// TIA Portal V19 export
FUNCTION "OUTPUT" : Void   // FC2, LAD
{ S7_Optimized_Access := 'TRUE' }
// stored: SetENOAutomatically false
BEGIN

REGION Network 1: "MFG FEED PUMP OP"
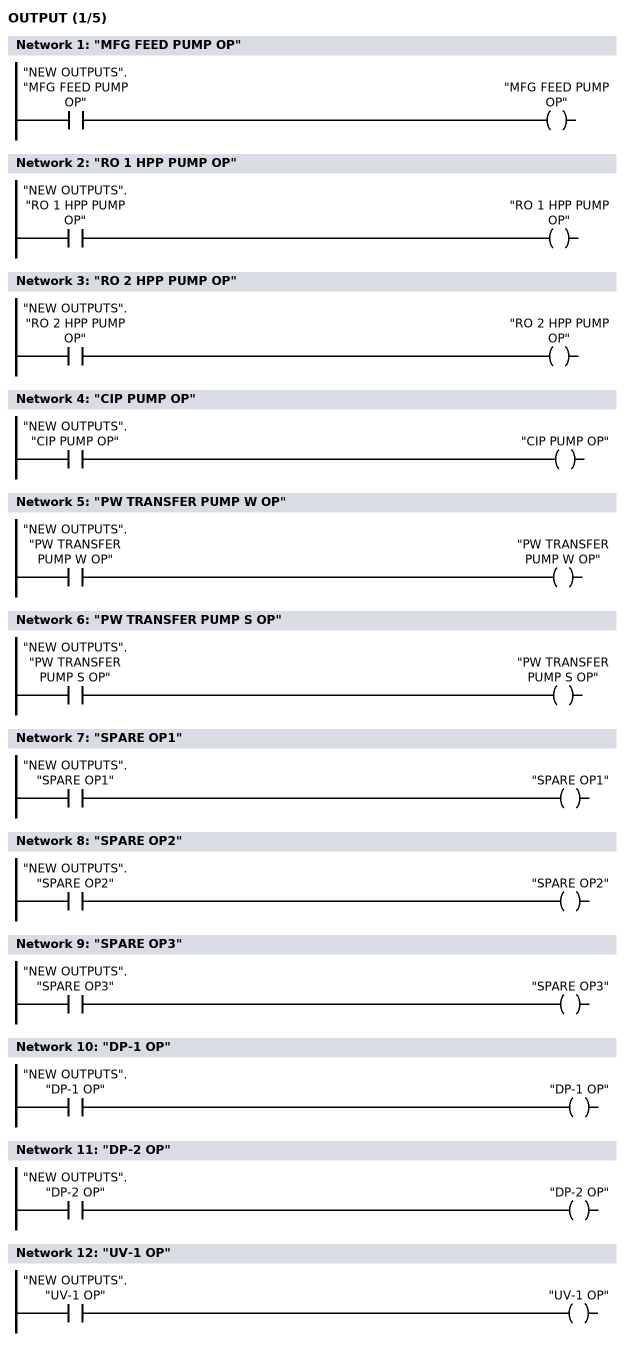
   RUNG wire#powerrail
      Contact( "NEW OUTPUTS"."MFG FEED PUMP OP" )
      Coil( "MFG FEED PUMP OP" )
   END_RUNG
   // the same network as SCL:
   "MFG FEED PUMP OP" := "NEW OUTPUTS"."MFG FEED PUMP OP";
END_REGION

REGION Network 2: "RO 1 HPP PUMP OP"
   RUNG wire#powerrail
      Contact( "NEW OUTPUTS"."RO 1 HPP PUMP OP" )
      Coil( "RO 1 HPP PUMP OP" )
   END_RUNG
   // the same network as SCL:
   "RO 1 HPP PUMP OP" := "NEW OUTPUTS"."RO 1 HPP PUMP OP";
END_REGION

REGION Network 3: "RO 2 HPP PUMP OP"
   RUNG wire#powerrail
      Contact( "NEW OUTPUTS"."RO 2 HPP PUMP OP" )
      Coil( "RO 2 HPP PUMP OP" )
   END_RUNG
   // the same network as SCL:
   "RO 2 HPP PUMP OP" := "NEW OUTPUTS"."RO 2 HPP PUMP OP";
END_REGION

REGION Network 4: "CIP PUMP OP"
   RUNG wire#powerrail
      Contact( "NEW OUTPUTS"."CIP PUMP OP" )
      Coil( "CIP PUMP OP" )
   END_RUNG
   // the same network as SCL:
   "CIP PUMP OP" := "NEW OUTPUTS"."CIP PUMP OP";
END_REGION

REGION Network 5: "PW TRANSFER PUMP W OP"
   RUNG wire#powerrail
      Contact( "NEW OUTPUTS"."PW TRANSFER PUMP W OP" )
      Coil( "PW TRANSFER PUMP W OP" )
   END_RUNG
   // the same network as SCL:
   "PW TRANSFER PUMP W OP" := "NEW OUTPUTS"."PW TRANSFER PUMP W OP";
END_REGION

REGION Network 6: "PW TRANSFER PUMP S OP"
   RUNG wire#powerrail
      Contact( "NEW OUTPUTS"."PW TRANSFER PUMP S OP" )
      Coil( "PW TRANSFER PUMP S OP" )
   END_RUNG
   // the same network as SCL:
   "PW TRANSFER PUMP S OP" := "NEW OUTPUTS"."PW TRANSFER PUMP S OP";
END_REGION

REGION Network 7: "SPARE OP1"
   RUNG wire#powerrail
      Contact( "NEW OUTPUTS"."SPARE OP1" )
      Coil( "SPARE OP1" )
   END_RUNG
   // the same network as SCL:
   "SPARE OP1" := "NEW OUTPUTS"."SPARE OP1";
END_REGION

REGION Network 8: "SPARE OP2"
   RUNG wire#powerrail
      Contact( "NEW OUTPUTS"."SPARE OP2" )
      Coil( "SPARE OP2" )
   END_RUNG
   // the same network as SCL:
   "SPARE OP2" := "NEW OUTPUTS"."SPARE OP2";
END_REGION

REGION Network 9: "SPARE OP3"
   RUNG wire#powerrail
      Contact( "NEW OUTPUTS"."SPARE OP3" )
      Coil( "SPARE OP3" )
   END_RUNG
   // the same network as SCL:
   "SPARE OP3" := "NEW OUTPUTS"."SPARE OP3";
END_REGION

REGION Network 10: "DP-1 OP"
   RUNG wire#powerrail
      Contact( "NEW OUTPUTS"."DP-1 OP" )
      Coil( "DP-1 OP" )
   END_RUNG
   // the same network as SCL:
   "DP-1 OP" := "NEW OUTPUTS"."DP-1 OP";
END_REGION

REGION Network 11: "DP-2 OP"
   RUNG wire#powerrail
      Contact( "NEW OUTPUTS"."DP-2 OP" )
      Coil( "DP-2 OP" )
   END_RUNG
   // the same network as SCL:
   "DP-2 OP" := "NEW OUTPUTS"."DP-2 OP";
END_REGION

REGION Network 12: "UV-1 OP"
   RUNG wire#powerrail
      Contact( "NEW OUTPUTS"."UV-1 OP" )
      Coil( "UV-1 OP" )
   END_RUNG
   // the same network as SCL:
   "UV-1 OP" := "NEW OUTPUTS"."UV-1 OP";
END_REGION

REGION Network 13: "SPARE OP4"
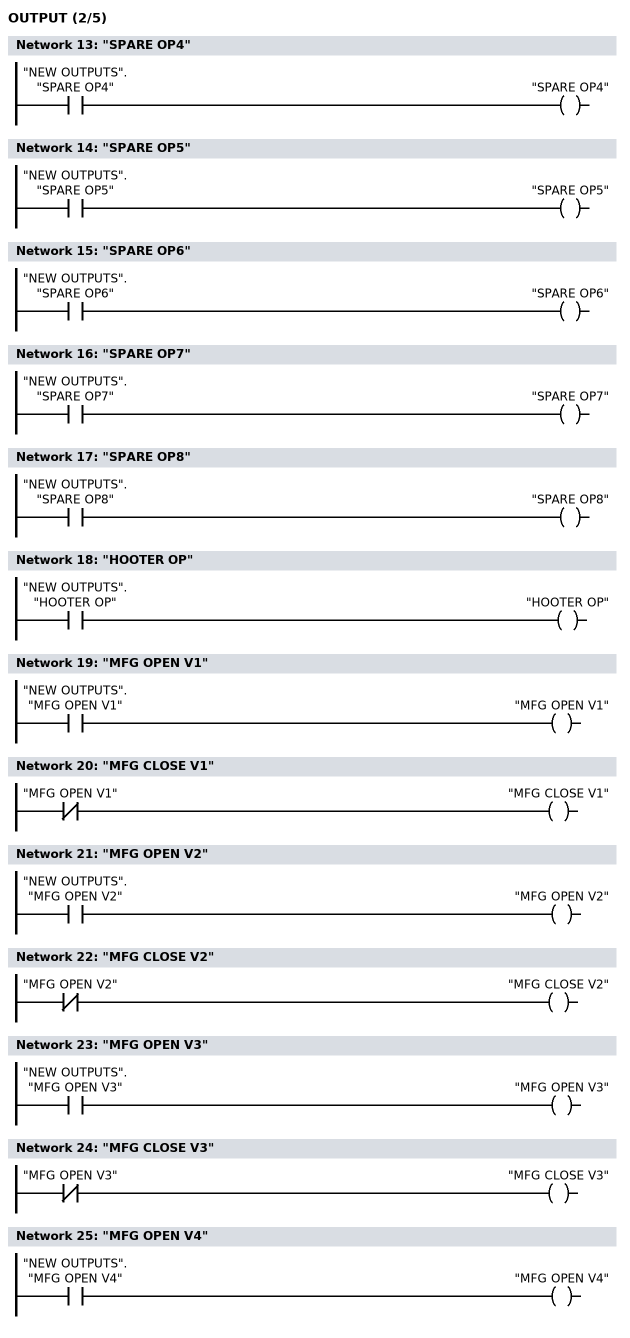
   RUNG wire#powerrail
      Contact( "NEW OUTPUTS"."SPARE OP4" )
      Coil( "SPARE OP4" )
   END_RUNG
   // the same network as SCL:
   "SPARE OP4" := "NEW OUTPUTS"."SPARE OP4";
END_REGION

REGION Network 14: "SPARE OP5"
   RUNG wire#powerrail
      Contact( "NEW OUTPUTS"."SPARE OP5" )
      Coil( "SPARE OP5" )
   END_RUNG
   // the same network as SCL:
   "SPARE OP5" := "NEW OUTPUTS"."SPARE OP5";
END_REGION

REGION Network 15: "SPARE OP6"
   RUNG wire#powerrail
      Contact( "NEW OUTPUTS"."SPARE OP6" )
      Coil( "SPARE OP6" )
   END_RUNG
   // the same network as SCL:
   "SPARE OP6" := "NEW OUTPUTS"."SPARE OP6";
END_REGION

REGION Network 16: "SPARE OP7"
   RUNG wire#powerrail
      Contact( "NEW OUTPUTS"."SPARE OP7" )
      Coil( "SPARE OP7" )
   END_RUNG
   // the same network as SCL:
   "SPARE OP7" := "NEW OUTPUTS"."SPARE OP7";
END_REGION

REGION Network 17: "SPARE OP8"
   RUNG wire#powerrail
      Contact( "NEW OUTPUTS"."SPARE OP8" )
      Coil( "SPARE OP8" )
   END_RUNG
   // the same network as SCL:
   "SPARE OP8" := "NEW OUTPUTS"."SPARE OP8";
END_REGION

REGION Network 18: "HOOTER OP"
   RUNG wire#powerrail
      Contact( "NEW OUTPUTS"."HOOTER OP" )
      Coil( "HOOTER OP" )
   END_RUNG
   // the same network as SCL:
   "HOOTER OP" := "NEW OUTPUTS"."HOOTER OP";
END_REGION

REGION Network 19: "MFG OPEN V1"
   RUNG wire#powerrail
      Contact( "NEW OUTPUTS"."MFG OPEN V1" )
      Coil( "MFG OPEN V1" )
   END_RUNG
   // the same network as SCL:
   "MFG OPEN V1" := "NEW OUTPUTS"."MFG OPEN V1";
END_REGION

REGION Network 20: "MFG CLOSE V1"
   RUNG wire#powerrail
      I_Contact( "MFG OPEN V1" )
      Coil( "MFG CLOSE V1" )
   END_RUNG
   // the same network as SCL:
   "MFG CLOSE V1" := NOT "MFG OPEN V1";
END_REGION

REGION Network 21: "MFG OPEN V2"
   RUNG wire#powerrail
      Contact( "NEW OUTPUTS"."MFG OPEN V2" )
      Coil( "MFG OPEN V2" )
   END_RUNG
   // the same network as SCL:
   "MFG OPEN V2" := "NEW OUTPUTS"."MFG OPEN V2";
END_REGION

REGION Network 22: "MFG CLOSE V2"
   RUNG wire#powerrail
      I_Contact( "MFG OPEN V2" )
      Coil( "MFG CLOSE V2" )
   END_RUNG
   // the same network as SCL:
   "MFG CLOSE V2" := NOT "MFG OPEN V2";
END_REGION

REGION Network 23: "MFG OPEN V3"
   RUNG wire#powerrail
      Contact( "NEW OUTPUTS"."MFG OPEN V3" )
      Coil( "MFG OPEN V3" )
   END_RUNG
   // the same network as SCL:
   "MFG OPEN V3" := "NEW OUTPUTS"."MFG OPEN V3";
END_REGION

REGION Network 24: "MFG CLOSE V3"
   RUNG wire#powerrail
      I_Contact( "MFG OPEN V3" )
      Coil( "MFG CLOSE V3" )
   END_RUNG
   // the same network as SCL:
   "MFG CLOSE V3" := NOT "MFG OPEN V3";
END_REGION

REGION Network 25: "MFG OPEN V4"
   RUNG wire#powerrail
      Contact( "NEW OUTPUTS"."MFG OPEN V4" )
      Coil( "MFG OPEN V4" )
   END_RUNG
   // the same network as SCL:
   "MFG OPEN V4" := "NEW OUTPUTS"."MFG OPEN V4";
END_REGION

REGION Network 26: "MFG CLOSE V4"
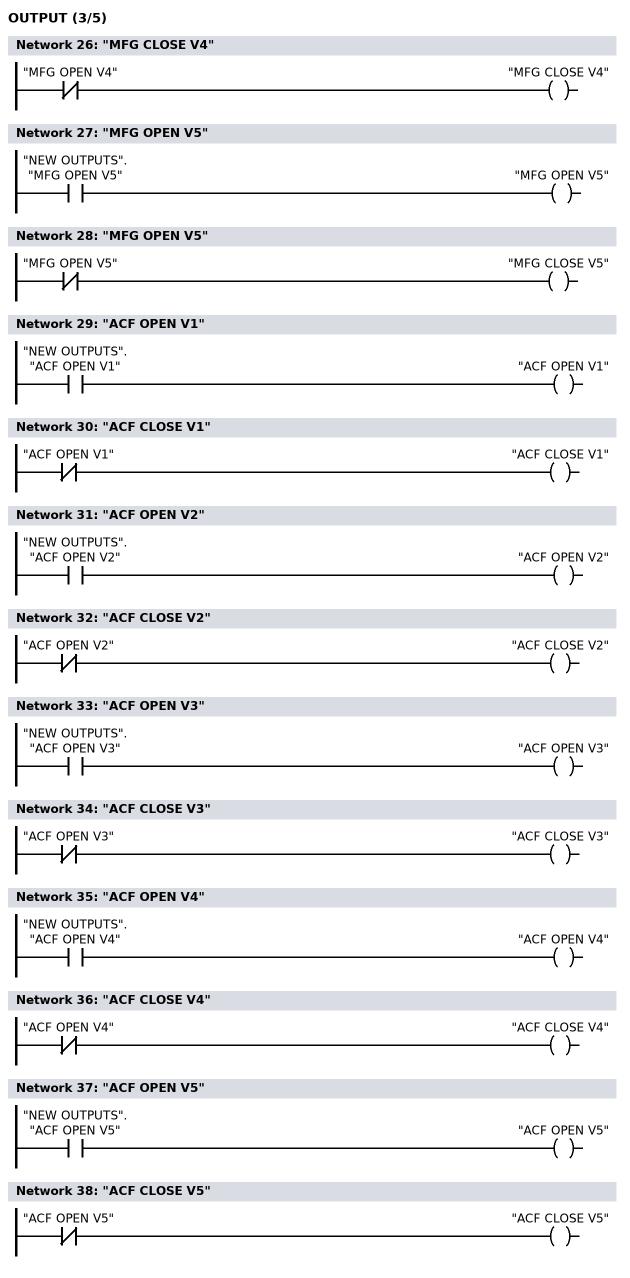
   RUNG wire#powerrail
      I_Contact( "MFG OPEN V4" )
      Coil( "MFG CLOSE V4" )
   END_RUNG
   // the same network as SCL:
   "MFG CLOSE V4" := NOT "MFG OPEN V4";
END_REGION

REGION Network 27: "MFG OPEN V5"
   RUNG wire#powerrail
      Contact( "NEW OUTPUTS"."MFG OPEN V5" )
      Coil( "MFG OPEN V5" )
   END_RUNG
   // the same network as SCL:
   "MFG OPEN V5" := "NEW OUTPUTS"."MFG OPEN V5";
END_REGION

REGION Network 28: "MFG OPEN V5"
   RUNG wire#powerrail
      I_Contact( "MFG OPEN V5" )
      Coil( "MFG CLOSE V5" )
   END_RUNG
   // the same network as SCL:
   "MFG CLOSE V5" := NOT "MFG OPEN V5";
END_REGION

REGION Network 29: "ACF OPEN V1"
   RUNG wire#powerrail
      Contact( "NEW OUTPUTS"."ACF OPEN V1" )
      Coil( "ACF OPEN V1" )
   END_RUNG
   // the same network as SCL:
   "ACF OPEN V1" := "NEW OUTPUTS"."ACF OPEN V1";
END_REGION

REGION Network 30: "ACF CLOSE V1"
   RUNG wire#powerrail
      I_Contact( "ACF OPEN V1" )
      Coil( "ACF CLOSE V1" )
   END_RUNG
   // the same network as SCL:
   "ACF CLOSE V1" := NOT "ACF OPEN V1";
END_REGION

REGION Network 31: "ACF OPEN V2"
   RUNG wire#powerrail
      Contact( "NEW OUTPUTS"."ACF OPEN V2" )
      Coil( "ACF OPEN V2" )
   END_RUNG
   // the same network as SCL:
   "ACF OPEN V2" := "NEW OUTPUTS"."ACF OPEN V2";
END_REGION

REGION Network 32: "ACF CLOSE V2"
   RUNG wire#powerrail
      I_Contact( "ACF OPEN V2" )
      Coil( "ACF CLOSE V2" )
   END_RUNG
   // the same network as SCL:
   "ACF CLOSE V2" := NOT "ACF OPEN V2";
END_REGION

REGION Network 33: "ACF OPEN V3"
   RUNG wire#powerrail
      Contact( "NEW OUTPUTS"."ACF OPEN V3" )
      Coil( "ACF OPEN V3" )
   END_RUNG
   // the same network as SCL:
   "ACF OPEN V3" := "NEW OUTPUTS"."ACF OPEN V3";
END_REGION

REGION Network 34: "ACF CLOSE V3"
   RUNG wire#powerrail
      I_Contact( "ACF OPEN V3" )
      Coil( "ACF CLOSE V3" )
   END_RUNG
   // the same network as SCL:
   "ACF CLOSE V3" := NOT "ACF OPEN V3";
END_REGION

REGION Network 35: "ACF OPEN V4"
   RUNG wire#powerrail
      Contact( "NEW OUTPUTS"."ACF OPEN V4" )
      Coil( "ACF OPEN V4" )
   END_RUNG
   // the same network as SCL:
   "ACF OPEN V4" := "NEW OUTPUTS"."ACF OPEN V4";
END_REGION

REGION Network 36: "ACF CLOSE V4"
   RUNG wire#powerrail
      I_Contact( "ACF OPEN V4" )
      Coil( "ACF CLOSE V4" )
   END_RUNG
   // the same network as SCL:
   "ACF CLOSE V4" := NOT "ACF OPEN V4";
END_REGION

REGION Network 37: "ACF OPEN V5"
   RUNG wire#powerrail
      Contact( "NEW OUTPUTS"."ACF OPEN V5" )
      Coil( "ACF OPEN V5" )
   END_RUNG
   // the same network as SCL:
   "ACF OPEN V5" := "NEW OUTPUTS"."ACF OPEN V5";
END_REGION

REGION Network 38: "ACF CLOSE V5"
   RUNG wire#powerrail
      I_Contact( "ACF OPEN V5" )
      Coil( "ACF CLOSE V5" )
   END_RUNG
   // the same network as SCL:
   "ACF CLOSE V5" := NOT "ACF OPEN V5";
END_REGION

REGION Network 39: "SF OPEN V1"
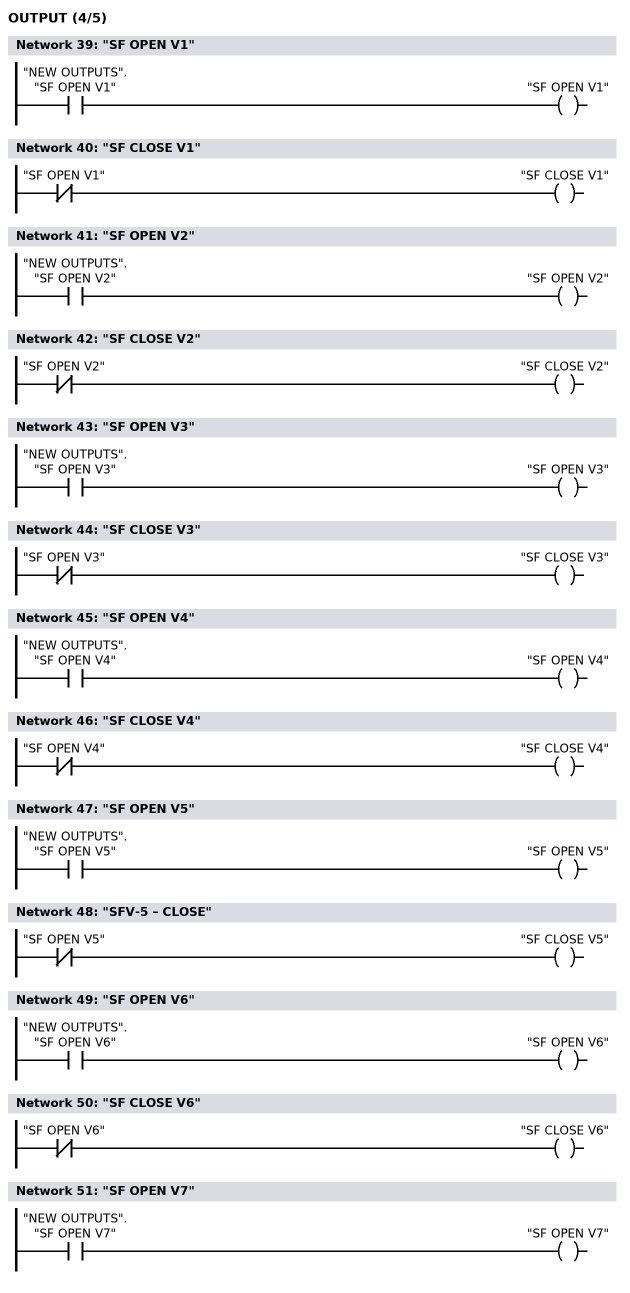
   RUNG wire#powerrail
      Contact( "NEW OUTPUTS"."SF OPEN V1" )
      Coil( "SF OPEN V1" )
   END_RUNG
   // the same network as SCL:
   "SF OPEN V1" := "NEW OUTPUTS"."SF OPEN V1";
END_REGION

REGION Network 40: "SF CLOSE V1"
   RUNG wire#powerrail
      I_Contact( "SF OPEN V1" )
      Coil( "SF CLOSE V1" )
   END_RUNG
   // the same network as SCL:
   "SF CLOSE V1" := NOT "SF OPEN V1";
END_REGION

REGION Network 41: "SF OPEN V2"
   RUNG wire#powerrail
      Contact( "NEW OUTPUTS"."SF OPEN V2" )
      Coil( "SF OPEN V2" )
   END_RUNG
   // the same network as SCL:
   "SF OPEN V2" := "NEW OUTPUTS"."SF OPEN V2";
END_REGION

REGION Network 42: "SF CLOSE V2"
   RUNG wire#powerrail
      I_Contact( "SF OPEN V2" )
      Coil( "SF CLOSE V2" )
   END_RUNG
   // the same network as SCL:
   "SF CLOSE V2" := NOT "SF OPEN V2";
END_REGION

REGION Network 43: "SF OPEN V3"
   RUNG wire#powerrail
      Contact( "NEW OUTPUTS"."SF OPEN V3" )
      Coil( "SF OPEN V3" )
   END_RUNG
   // the same network as SCL:
   "SF OPEN V3" := "NEW OUTPUTS"."SF OPEN V3";
END_REGION

REGION Network 44: "SF CLOSE V3"
   RUNG wire#powerrail
      I_Contact( "SF OPEN V3" )
      Coil( "SF CLOSE V3" )
   END_RUNG
   // the same network as SCL:
   "SF CLOSE V3" := NOT "SF OPEN V3";
END_REGION

REGION Network 45: "SF OPEN V4"
   RUNG wire#powerrail
      Contact( "NEW OUTPUTS"."SF OPEN V4" )
      Coil( "SF OPEN V4" )
   END_RUNG
   // the same network as SCL:
   "SF OPEN V4" := "NEW OUTPUTS"."SF OPEN V4";
END_REGION

REGION Network 46: "SF CLOSE V4"
   RUNG wire#powerrail
      I_Contact( "SF OPEN V4" )
      Coil( "SF CLOSE V4" )
   END_RUNG
   // the same network as SCL:
   "SF CLOSE V4" := NOT "SF OPEN V4";
END_REGION

REGION Network 47: "SF OPEN V5"
   RUNG wire#powerrail
      Contact( "NEW OUTPUTS"."SF OPEN V5" )
      Coil( "SF OPEN V5" )
   END_RUNG
   // the same network as SCL:
   "SF OPEN V5" := "NEW OUTPUTS"."SF OPEN V5";
END_REGION

REGION Network 48: "SFV-5 – CLOSE"
   RUNG wire#powerrail
      I_Contact( "SF OPEN V5" )
      Coil( "SF CLOSE V5" )
   END_RUNG
   // the same network as SCL:
   "SF CLOSE V5" := NOT "SF OPEN V5";
END_REGION

REGION Network 49: "SF OPEN V6"
   RUNG wire#powerrail
      Contact( "NEW OUTPUTS"."SF OPEN V6" )
      Coil( "SF OPEN V6" )
   END_RUNG
   // the same network as SCL:
   "SF OPEN V6" := "NEW OUTPUTS"."SF OPEN V6";
END_REGION

REGION Network 50: "SF CLOSE V6"
   RUNG wire#powerrail
      I_Contact( "SF OPEN V6" )
      Coil( "SF CLOSE V6" )
   END_RUNG
   // the same network as SCL:
   "SF CLOSE V6" := NOT "SF OPEN V6";
END_REGION

REGION Network 51: "SF OPEN V7"
   RUNG wire#powerrail
      Contact( "NEW OUTPUTS"."SF OPEN V7" )
      Coil( "SF OPEN V7" )
   END_RUNG
   // the same network as SCL:
   "SF OPEN V7" := "NEW OUTPUTS"."SF OPEN V7";
END_REGION

REGION Network 52: "SF CLOSE V7"
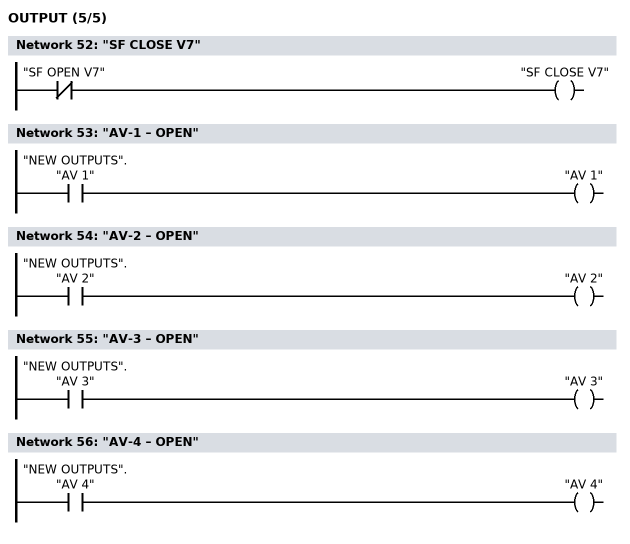
   RUNG wire#powerrail
      I_Contact( "SF OPEN V7" )
      Coil( "SF CLOSE V7" )
   END_RUNG
   // the same network as SCL:
   "SF CLOSE V7" := NOT "SF OPEN V7";
END_REGION

REGION Network 53: "AV-1 – OPEN"
   RUNG wire#powerrail
      Contact( "NEW OUTPUTS"."AV 1" )
      Coil( "AV 1" )
   END_RUNG
   // the same network as SCL:
   "AV 1" := "NEW OUTPUTS"."AV 1";
END_REGION

REGION Network 54: "AV-2 – OPEN"
   RUNG wire#powerrail
      Contact( "NEW OUTPUTS"."AV 2" )
      Coil( "AV 2" )
   END_RUNG
   // the same network as SCL:
   "AV 2" := "NEW OUTPUTS"."AV 2";
END_REGION

REGION Network 55: "AV-3 – OPEN"
   RUNG wire#powerrail
      Contact( "NEW OUTPUTS"."AV 3" )
      Coil( "AV 3" )
   END_RUNG
   // the same network as SCL:
   "AV 3" := "NEW OUTPUTS"."AV 3";
END_REGION

REGION Network 56: "AV-4 – OPEN"
   RUNG wire#powerrail
      Contact( "NEW OUTPUTS"."AV 4" )
      Coil( "AV 4" )
   END_RUNG
   // the same network as SCL:
   "AV 4" := "NEW OUTPUTS"."AV 4";
END_REGION
END_FUNCTION
